Fanuc KAREL source: kt00524.KL

-- PROVISIONAL review KL for V770-1; original PC SHA256 bafe0d1d8a31af757d8c7888787d8f3ae3f65d339f0726742d2c5a02ff79dc8e
-- Incomplete behavior may be omitted. Consult companion uncertainty JSON. Do not deploy.
PROGRAM KT00524
%NOLOCKGROUP
-- UNRESOLVED_DECL P1 type=000106
-- UNRESOLVED_DECL P2 type=000106
-- UNRESOLVED_DECL OUT type=000101
BEGIN
  -- UNRESOLVED_PC offsets 5-20; opcodes 2E,22,32,35
  -- UNRESOLVED_PC offsets 25-40; opcodes 2E,22,32,35
  -- UNRESOLVED_PC offsets 45-60; opcodes 2E,22,32,35
  -- UNRESOLVED_PC offsets 65-80; opcodes 2E,22,32,35
  -- UNRESOLVED_PC offsets 85-119; opcodes 49,7E,49,7E,60,4A
  -- UNRESOLVED_PC offsets 124-128; opcodes 7F
END KT00524
